// TIA Portal V20 export
TYPE "type_emRelations_em4"
// stored: Access Published, Namespace Unit1
   STRUCT
      "Bool" { ExternalWritable := 'False'} : Array[0..99] of Bool;
      LReal { ExternalWritable := 'False'} : Array[0..19] of LReal;
      isLinked { ExternalWritable := 'False'} : Bool;
      softCam { ExternalWritable := 'False'} : "Unit1.type_emRelations_em4_SoftCam";
      cmControlNode { ExternalWritable := 'False'} : "Unit1.type_emRelations_em4_cmStatus";
      cmConfig { ExternalWritable := 'False'} : Struct
         cmAnodeMainPnP1AxisX : "LBC_typeAxis64PosConfiguration";
      END_STRUCT;
      sequence { ExternalWritable := 'False'} : "Unit1.type_emRelations_em4_sequence";
   END_STRUCT;
END_TYPE
